TYPE ST_CAMERA_Mapping :
STRUCT
	nIndex				: INT;
	nReqProgram			: BYTE;
	aPackPos			: ARRAY[1..5, 1..cMAX_CAMERA_PROG_NUMBER] OF BYTE;
	aTargetBuffer		: ARRAY[1..5] OF BYTE;

END_STRUCT
END_TYPE

(* stored: Version 1.1.0.1
   DUT ST_CAMERA_Mapping: Id {87ad718d-a03a-4c0f-9dc8-ebda85a0a3fb} *)
